// TIA Portal V20 export
ORGANIZATION_BLOCK "Startup"   // OB1000, LAD, Startup
TITLE = "Complete Restart"
AUTHOR : ERsystem_FA2_DH. Kim
// stored: AutoNumber false, IsIECCheckEnabled true, Namespace Unit1, SetENOAutomatically false
   VAR_INPUT
      LostRetentive : Bool;   // True if retentive data are lost
      LostRTC : Bool;   // True if date and time are lost
   END_VAR
   VAR_TEMP
      tempIndex : Int;   // Index of Unit in the array
   END_VAR
BEGIN

REGION Network 1: Unit Index Number
   // Assign the number of the unit to a temp for correct array index access.
   // Number is defined in PLC tags of Software Unit Global.
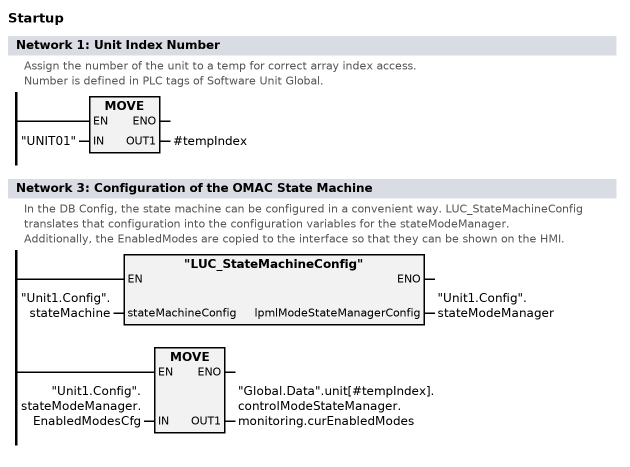
   RUNG wire#powerrail
      Move(in := "UNIT01", out1 => #tempIndex)
   END_RUNG
   // the same network as SCL:
   #tempIndex := "UNIT01";
END_REGION

REGION Network 2 (SCL): Build the Absolut Reference Designator
   // Set the Absoult Reference Designator in the DB Config. It is combined out of the parent reference designator and the own reference designator (=relative)
   IF LEN(IN := "Unit1.Config".unit.referenceDesignator.parent) <> 0 THEN
     "Unit1.Config".unit.referenceDesignator.combined := CONCAT_WSTRING(IN1 := "Unit1.Config".unit.referenceDesignator.parent, IN2 := WSTRING#'.', IN3 := "Unit1.Config".unit.referenceDesignator.relative);
   ELSE
     "Unit1.Config".unit.referenceDesignator.combined := "Unit1.Config".unit.referenceDesignator.relative;
   END_IF;
END_REGION

REGION Network 3: Configuration of the OMAC State Machine
   // In the DB Config, the state machine can be configured in a convenient way. LUC_StateMachineConfig translates that configuration into the configuration variables for the stateModeManager.
   // Additionally, the EnabledModes are copied to the interface so that they can be shown on the HMI.
   RUNG wire#powerrail
      "LUC_StateMachineConfig"(stateMachineConfig := "Unit1.Config".stateMachine, lpmlModeStateManagerConfig => "Unit1.Config".stateModeManager)
   END_RUNG
   RUNG wire#powerrail
      Move(in := "Unit1.Config".stateModeManager.EnabledModesCfg, out1 => "Global.Data".unit[#tempIndex].controlModeStateManager.monitoring.curEnabledModes)
   END_RUNG
   // the same network as SCL:
   "LUC_StateMachineConfig"(stateMachineConfig := "Unit1.Config".stateMachine,
                           lpmlModeStateManagerConfig => "Unit1.Config".stateModeManager);
   "Global.Data".unit[#tempIndex].controlModeStateManager.monitoring.curEnabledModes := "Unit1.Config".stateModeManager.EnabledModesCfg;
END_REGION

REGION Network 4 (SCL): Configuration of Stack Light
   // undefined
   "Unit1.Config".signalStack.undefined.static.red := FALSE;
   "Unit1.Config".signalStack.undefined.static.yellow := FALSE;
   "Unit1.Config".signalStack.undefined.static.blue := FALSE;
   "Unit1.Config".signalStack.undefined.static.green := FALSE;
   "Unit1.Config".signalStack.undefined.static.horn := FALSE;
   "Unit1.Config".signalStack.undefined.static.white := FALSE;
   "Unit1.Config".signalStack.undefined.static.user1 := FALSE;
   "Unit1.Config".signalStack.undefined.static.user2 := FALSE;

   "Unit1.Config".signalStack.undefined.flashing.red := TRUE;
   "Unit1.Config".signalStack.undefined.flashing.yellow := FALSE;
   "Unit1.Config".signalStack.undefined.flashing.blue := FALSE;
   "Unit1.Config".signalStack.undefined.flashing.green := FALSE;
   "Unit1.Config".signalStack.undefined.flashing.horn := FALSE;
   "Unit1.Config".signalStack.undefined.flashing.white := FALSE;
   "Unit1.Config".signalStack.undefined.flashing.user1 := FALSE;
   "Unit1.Config".signalStack.undefined.flashing.user2 := FALSE;

   // clearing
   "Unit1.Config".signalStack.clearing.static.red := FALSE;
   "Unit1.Config".signalStack.clearing.static.yellow := FALSE;
   "Unit1.Config".signalStack.clearing.static.blue := FALSE;
   "Unit1.Config".signalStack.clearing.static.green := FALSE;
   "Unit1.Config".signalStack.clearing.static.horn := FALSE;
   "Unit1.Config".signalStack.clearing.static.white := FALSE;
   "Unit1.Config".signalStack.clearing.static.user1 := FALSE;
   "Unit1.Config".signalStack.clearing.static.user2 := FALSE;

   "Unit1.Config".signalStack.clearing.flashing.red := TRUE;
   "Unit1.Config".signalStack.clearing.flashing.yellow := FALSE;
   "Unit1.Config".signalStack.clearing.flashing.blue := FALSE;
   "Unit1.Config".signalStack.clearing.flashing.green := FALSE;
   "Unit1.Config".signalStack.clearing.flashing.horn := FALSE;
   "Unit1.Config".signalStack.clearing.flashing.white := FALSE;
   "Unit1.Config".signalStack.clearing.flashing.user1 := FALSE;
   "Unit1.Config".signalStack.clearing.flashing.user2 := FALSE;

   // stopped
   "Unit1.Config".signalStack.stopped.static.red := TRUE;
   "Unit1.Config".signalStack.stopped.static.yellow := FALSE;
   "Unit1.Config".signalStack.stopped.static.blue := FALSE;
   "Unit1.Config".signalStack.stopped.static.green := FALSE;
   "Unit1.Config".signalStack.stopped.static.horn := FALSE;
   "Unit1.Config".signalStack.stopped.static.white := FALSE;
   "Unit1.Config".signalStack.stopped.static.user1 := FALSE;
   "Unit1.Config".signalStack.stopped.static.user2 := FALSE;

   "Unit1.Config".signalStack.stopped.flashing.red := FALSE;
   "Unit1.Config".signalStack.stopped.flashing.yellow := FALSE;
   "Unit1.Config".signalStack.stopped.flashing.blue := FALSE;
   "Unit1.Config".signalStack.stopped.flashing.green := FALSE;
   "Unit1.Config".signalStack.stopped.flashing.horn := FALSE;
   "Unit1.Config".signalStack.stopped.flashing.white := FALSE;
   "Unit1.Config".signalStack.stopped.flashing.user1 := FALSE;
   "Unit1.Config".signalStack.stopped.flashing.user2 := FALSE;

   // starting
   "Unit1.Config".signalStack.starting.static.red := FALSE;
   "Unit1.Config".signalStack.starting.static.yellow := FALSE;
   "Unit1.Config".signalStack.starting.static.blue := FALSE;
   "Unit1.Config".signalStack.starting.static.green := TRUE;
   "Unit1.Config".signalStack.starting.static.horn := FALSE;
   "Unit1.Config".signalStack.starting.static.white := FALSE;
   "Unit1.Config".signalStack.starting.static.user1 := FALSE;
   "Unit1.Config".signalStack.starting.static.user2 := FALSE;

   "Unit1.Config".signalStack.starting.flashing.red := FALSE;
   "Unit1.Config".signalStack.starting.flashing.yellow := FALSE;
   "Unit1.Config".signalStack.starting.flashing.blue := FALSE;
   "Unit1.Config".signalStack.starting.flashing.green := FALSE;
   "Unit1.Config".signalStack.starting.flashing.horn := FALSE;
   "Unit1.Config".signalStack.starting.flashing.white := FALSE;
   "Unit1.Config".signalStack.starting.flashing.user1 := FALSE;
   "Unit1.Config".signalStack.starting.flashing.user2 := FALSE;

   // idle
   "Unit1.Config".signalStack.idle.static.red := FALSE;
   "Unit1.Config".signalStack.idle.static.yellow := FALSE;
   "Unit1.Config".signalStack.idle.static.blue := FALSE;
   "Unit1.Config".signalStack.idle.static.green := FALSE;
   "Unit1.Config".signalStack.idle.static.horn := FALSE;
   "Unit1.Config".signalStack.idle.static.white := FALSE;
   "Unit1.Config".signalStack.idle.static.user1 := FALSE;
   "Unit1.Config".signalStack.idle.static.user2 := FALSE;

   "Unit1.Config".signalStack.idle.flashing.red := FALSE;
   "Unit1.Config".signalStack.idle.flashing.yellow := FALSE;
   "Unit1.Config".signalStack.idle.flashing.blue := FALSE;
   "Unit1.Config".signalStack.idle.flashing.green := TRUE;
   "Unit1.Config".signalStack.idle.flashing.horn := FALSE;
   "Unit1.Config".signalStack.idle.flashing.white := FALSE;
   "Unit1.Config".signalStack.idle.flashing.user1 := FALSE;
   "Unit1.Config".signalStack.idle.flashing.user2 := FALSE;

   // suspended
   "Unit1.Config".signalStack.suspended.static.red := FALSE;
   "Unit1.Config".signalStack.suspended.static.yellow := TRUE;
   "Unit1.Config".signalStack.suspended.static.blue := FALSE;
   "Unit1.Config".signalStack.suspended.static.green := FALSE;
   "Unit1.Config".signalStack.suspended.static.horn := FALSE;
   "Unit1.Config".signalStack.suspended.static.white := FALSE;
   "Unit1.Config".signalStack.suspended.static.user1 := FALSE;
   "Unit1.Config".signalStack.suspended.static.user2 := FALSE;

   "Unit1.Config".signalStack.suspended.flashing.red := FALSE;
   "Unit1.Config".signalStack.suspended.flashing.yellow := FALSE;
   "Unit1.Config".signalStack.suspended.flashing.blue := FALSE;
   "Unit1.Config".signalStack.suspended.flashing.green := FALSE;
   "Unit1.Config".signalStack.suspended.flashing.horn := FALSE;
   "Unit1.Config".signalStack.suspended.flashing.white := FALSE;
   "Unit1.Config".signalStack.suspended.flashing.user1 := FALSE;
   "Unit1.Config".signalStack.suspended.flashing.user2 := FALSE;

   // execute
   "Unit1.Config".signalStack.execute.static.red := FALSE;
   "Unit1.Config".signalStack.execute.static.yellow := FALSE;
   "Unit1.Config".signalStack.execute.static.blue := FALSE;
   "Unit1.Config".signalStack.execute.static.green := TRUE;
   "Unit1.Config".signalStack.execute.static.horn := FALSE;
   "Unit1.Config".signalStack.execute.static.white := FALSE;
   "Unit1.Config".signalStack.execute.static.user1 := FALSE;
   "Unit1.Config".signalStack.execute.static.user2 := FALSE;

   "Unit1.Config".signalStack.execute.flashing.red := FALSE;
   "Unit1.Config".signalStack.execute.flashing.yellow := FALSE;
   "Unit1.Config".signalStack.execute.flashing.blue := FALSE;
   "Unit1.Config".signalStack.execute.flashing.green := FALSE;
   "Unit1.Config".signalStack.execute.flashing.horn := FALSE;
   "Unit1.Config".signalStack.execute.flashing.white := FALSE;
   "Unit1.Config".signalStack.execute.flashing.user1 := FALSE;
   "Unit1.Config".signalStack.execute.flashing.user2 := FALSE;

   // stopping
   "Unit1.Config".signalStack.stopping.static.red := TRUE;
   "Unit1.Config".signalStack.stopping.static.yellow := FALSE;
   "Unit1.Config".signalStack.stopping.static.blue := FALSE;
   "Unit1.Config".signalStack.stopping.static.green := FALSE;
   "Unit1.Config".signalStack.stopping.static.horn := FALSE;
   "Unit1.Config".signalStack.stopping.static.white := FALSE;
   "Unit1.Config".signalStack.stopping.static.user1 := FALSE;
   "Unit1.Config".signalStack.stopping.static.user2 := FALSE;

   "Unit1.Config".signalStack.stopping.flashing.red := FALSE;
   "Unit1.Config".signalStack.stopping.flashing.yellow := FALSE;
   "Unit1.Config".signalStack.stopping.flashing.blue := FALSE;
   "Unit1.Config".signalStack.stopping.flashing.green := FALSE;
   "Unit1.Config".signalStack.stopping.flashing.horn := FALSE;
   "Unit1.Config".signalStack.stopping.flashing.white := FALSE;
   "Unit1.Config".signalStack.stopping.flashing.user1 := FALSE;
   "Unit1.Config".signalStack.stopping.flashing.user2 := FALSE;

   // aborting
   "Unit1.Config".signalStack.aborting.static.red := FALSE;
   "Unit1.Config".signalStack.aborting.static.yellow := FALSE;
   "Unit1.Config".signalStack.aborting.static.blue := FALSE;
   "Unit1.Config".signalStack.aborting.static.green := FALSE;
   "Unit1.Config".signalStack.aborting.static.horn := FALSE;
   "Unit1.Config".signalStack.aborting.static.white := FALSE;
   "Unit1.Config".signalStack.aborting.static.user1 := FALSE;
   "Unit1.Config".signalStack.aborting.static.user2 := FALSE;

   "Unit1.Config".signalStack.aborting.flashing.red := TRUE;
   "Unit1.Config".signalStack.aborting.flashing.yellow := FALSE;
   "Unit1.Config".signalStack.aborting.flashing.blue := FALSE;
   "Unit1.Config".signalStack.aborting.flashing.green := FALSE;
   "Unit1.Config".signalStack.aborting.flashing.horn := FALSE;
   "Unit1.Config".signalStack.aborting.flashing.white := FALSE;
   "Unit1.Config".signalStack.aborting.flashing.user1 := FALSE;
   "Unit1.Config".signalStack.aborting.flashing.user2 := FALSE;

   // aborted
   "Unit1.Config".signalStack.aborted.static.red := FALSE;
   "Unit1.Config".signalStack.aborted.static.yellow := FALSE;
   "Unit1.Config".signalStack.aborted.static.blue := FALSE;
   "Unit1.Config".signalStack.aborted.static.green := FALSE;
   "Unit1.Config".signalStack.aborted.static.horn := FALSE;
   "Unit1.Config".signalStack.aborted.static.white := FALSE;
   "Unit1.Config".signalStack.aborted.static.user1 := FALSE;
   "Unit1.Config".signalStack.aborted.static.user2 := FALSE;

   "Unit1.Config".signalStack.aborted.flashing.red := TRUE;
   "Unit1.Config".signalStack.aborted.flashing.yellow := FALSE;
   "Unit1.Config".signalStack.aborted.flashing.blue := FALSE;
   "Unit1.Config".signalStack.aborted.flashing.green := FALSE;
   "Unit1.Config".signalStack.aborted.flashing.horn := FALSE;
   "Unit1.Config".signalStack.aborted.flashing.white := FALSE;
   "Unit1.Config".signalStack.aborted.flashing.user1 := FALSE;
   "Unit1.Config".signalStack.aborted.flashing.user2 := FALSE;

   // holding
   "Unit1.Config".signalStack.holding.static.red := FALSE;
   "Unit1.Config".signalStack.holding.static.yellow := FALSE;
   "Unit1.Config".signalStack.holding.static.blue := FALSE;
   "Unit1.Config".signalStack.holding.static.green := FALSE;
   "Unit1.Config".signalStack.holding.static.horn := FALSE;
   "Unit1.Config".signalStack.holding.static.white := FALSE;
   "Unit1.Config".signalStack.holding.static.user1 := FALSE;
   "Unit1.Config".signalStack.holding.static.user2 := FALSE;

   "Unit1.Config".signalStack.holding.flashing.red := FALSE;
   "Unit1.Config".signalStack.holding.flashing.yellow := FALSE;
   "Unit1.Config".signalStack.holding.flashing.blue := TRUE;
   "Unit1.Config".signalStack.holding.flashing.green := FALSE;
   "Unit1.Config".signalStack.holding.flashing.horn := FALSE;
   "Unit1.Config".signalStack.holding.flashing.white := FALSE;
   "Unit1.Config".signalStack.holding.flashing.user1 := FALSE;
   "Unit1.Config".signalStack.holding.flashing.user2 := FALSE;

   // held
   "Unit1.Config".signalStack.held.static.red := FALSE;
   "Unit1.Config".signalStack.held.static.yellow := FALSE;
   "Unit1.Config".signalStack.held.static.blue := TRUE;
   "Unit1.Config".signalStack.held.static.green := FALSE;
   "Unit1.Config".signalStack.held.static.horn := FALSE;
   "Unit1.Config".signalStack.held.static.white := FALSE;
   "Unit1.Config".signalStack.held.static.user1 := FALSE;
   "Unit1.Config".signalStack.held.static.user2 := FALSE;

   "Unit1.Config".signalStack.held.flashing.red := FALSE;
   "Unit1.Config".signalStack.held.flashing.yellow := FALSE;
   "Unit1.Config".signalStack.held.flashing.blue := FALSE;
   "Unit1.Config".signalStack.held.flashing.green := FALSE;
   "Unit1.Config".signalStack.held.flashing.horn := FALSE;
   "Unit1.Config".signalStack.held.flashing.white := FALSE;
   "Unit1.Config".signalStack.held.flashing.user1 := FALSE;
   "Unit1.Config".signalStack.held.flashing.user2 := FALSE;

   // unholding
   "Unit1.Config".signalStack.unholding.static.red := FALSE;
   "Unit1.Config".signalStack.unholding.static.yellow := FALSE;
   "Unit1.Config".signalStack.unholding.static.blue := FALSE;
   "Unit1.Config".signalStack.unholding.static.green := TRUE;
   "Unit1.Config".signalStack.unholding.static.horn := FALSE;
   "Unit1.Config".signalStack.unholding.static.white := FALSE;
   "Unit1.Config".signalStack.unholding.static.user1 := FALSE;
   "Unit1.Config".signalStack.unholding.static.user2 := FALSE;

   "Unit1.Config".signalStack.unholding.flashing.red := FALSE;
   "Unit1.Config".signalStack.unholding.flashing.yellow := FALSE;
   "Unit1.Config".signalStack.unholding.flashing.blue := FALSE;
   "Unit1.Config".signalStack.unholding.flashing.green := FALSE;
   "Unit1.Config".signalStack.unholding.flashing.horn := FALSE;
   "Unit1.Config".signalStack.unholding.flashing.white := FALSE;
   "Unit1.Config".signalStack.unholding.flashing.user1 := FALSE;
   "Unit1.Config".signalStack.unholding.flashing.user2 := FALSE;

   // suspending
   "Unit1.Config".signalStack.suspending.static.red := FALSE;
   "Unit1.Config".signalStack.suspending.static.yellow := FALSE;
   "Unit1.Config".signalStack.suspending.static.blue := FALSE;
   "Unit1.Config".signalStack.suspending.static.green := FALSE;
   "Unit1.Config".signalStack.suspending.static.horn := FALSE;
   "Unit1.Config".signalStack.suspending.static.white := FALSE;
   "Unit1.Config".signalStack.suspending.static.user1 := FALSE;
   "Unit1.Config".signalStack.suspending.static.user2 := FALSE;

   "Unit1.Config".signalStack.suspending.flashing.red := FALSE;
   "Unit1.Config".signalStack.suspending.flashing.yellow := TRUE;
   "Unit1.Config".signalStack.suspending.flashing.blue := FALSE;
   "Unit1.Config".signalStack.suspending.flashing.green := FALSE;
   "Unit1.Config".signalStack.suspending.flashing.horn := FALSE;
   "Unit1.Config".signalStack.suspending.flashing.white := FALSE;
   "Unit1.Config".signalStack.suspending.flashing.user1 := FALSE;
   "Unit1.Config".signalStack.suspending.flashing.user2 := FALSE;

   // unsuspending
   "Unit1.Config".signalStack.unsuspending.static.red := FALSE;
   "Unit1.Config".signalStack.unsuspending.static.yellow := FALSE;
   "Unit1.Config".signalStack.unsuspending.static.blue := FALSE;
   "Unit1.Config".signalStack.unsuspending.static.green := TRUE;
   "Unit1.Config".signalStack.unsuspending.static.horn := FALSE;
   "Unit1.Config".signalStack.unsuspending.static.white := FALSE;
   "Unit1.Config".signalStack.unsuspending.static.user1 := FALSE;
   "Unit1.Config".signalStack.unsuspending.static.user2 := FALSE;

   "Unit1.Config".signalStack.unsuspending.flashing.red := FALSE;
   "Unit1.Config".signalStack.unsuspending.flashing.yellow := FALSE;
   "Unit1.Config".signalStack.unsuspending.flashing.blue := FALSE;
   "Unit1.Config".signalStack.unsuspending.flashing.green := FALSE;
   "Unit1.Config".signalStack.unsuspending.flashing.horn := FALSE;
   "Unit1.Config".signalStack.unsuspending.flashing.white := FALSE;
   "Unit1.Config".signalStack.unsuspending.flashing.user1 := FALSE;
   "Unit1.Config".signalStack.unsuspending.flashing.user2 := FALSE;

   // resetting
   "Unit1.Config".signalStack.resetting.static.red := TRUE;
   "Unit1.Config".signalStack.resetting.static.yellow := FALSE;
   "Unit1.Config".signalStack.resetting.static.blue := FALSE;
   "Unit1.Config".signalStack.resetting.static.green := FALSE;
   "Unit1.Config".signalStack.resetting.static.horn := FALSE;
   "Unit1.Config".signalStack.resetting.static.white := FALSE;
   "Unit1.Config".signalStack.resetting.static.user1 := FALSE;
   "Unit1.Config".signalStack.resetting.static.user2 := FALSE;

   "Unit1.Config".signalStack.resetting.flashing.red := FALSE;
   "Unit1.Config".signalStack.resetting.flashing.yellow := FALSE;
   "Unit1.Config".signalStack.resetting.flashing.blue := FALSE;
   "Unit1.Config".signalStack.resetting.flashing.green := FALSE;
   "Unit1.Config".signalStack.resetting.flashing.horn := FALSE;
   "Unit1.Config".signalStack.resetting.flashing.white := FALSE;
   "Unit1.Config".signalStack.resetting.flashing.user1 := FALSE;
   "Unit1.Config".signalStack.resetting.flashing.user2 := FALSE;

   // completing
   "Unit1.Config".signalStack.completing.static.red := FALSE;
   "Unit1.Config".signalStack.completing.static.yellow := FALSE;
   "Unit1.Config".signalStack.completing.static.blue := FALSE;
   "Unit1.Config".signalStack.completing.static.green := TRUE;
   "Unit1.Config".signalStack.completing.static.horn := FALSE;
   "Unit1.Config".signalStack.completing.static.white := FALSE;
   "Unit1.Config".signalStack.completing.static.user1 := FALSE;
   "Unit1.Config".signalStack.completing.static.user2 := FALSE;

   "Unit1.Config".signalStack.completing.flashing.red := FALSE;
   "Unit1.Config".signalStack.completing.flashing.yellow := FALSE;
   "Unit1.Config".signalStack.completing.flashing.blue := FALSE;
   "Unit1.Config".signalStack.completing.flashing.green := FALSE;
   "Unit1.Config".signalStack.completing.flashing.horn := FALSE;
   "Unit1.Config".signalStack.completing.flashing.white := FALSE;
   "Unit1.Config".signalStack.completing.flashing.user1 := FALSE;
   "Unit1.Config".signalStack.completing.flashing.user2 := FALSE;

   // completed
   "Unit1.Config".signalStack.completed.static.red := TRUE;
   "Unit1.Config".signalStack.completed.static.yellow := FALSE;
   "Unit1.Config".signalStack.completed.static.blue := FALSE;
   "Unit1.Config".signalStack.completed.static.green := FALSE;
   "Unit1.Config".signalStack.completed.static.horn := FALSE;
   "Unit1.Config".signalStack.completed.static.white := FALSE;
   "Unit1.Config".signalStack.completed.static.user1 := FALSE;
   "Unit1.Config".signalStack.completed.static.user2 := FALSE;

   "Unit1.Config".signalStack.completed.flashing.red := FALSE;
   "Unit1.Config".signalStack.completed.flashing.yellow := FALSE;
   "Unit1.Config".signalStack.completed.flashing.blue := FALSE;
   "Unit1.Config".signalStack.completed.flashing.green := FALSE;
   "Unit1.Config".signalStack.completed.flashing.horn := FALSE;
   "Unit1.Config".signalStack.completed.flashing.white := FALSE;
   "Unit1.Config".signalStack.completed.flashing.user1 := FALSE;
   "Unit1.Config".signalStack.completed.flashing.user2 := FALSE;
END_REGION
END_ORGANIZATION_BLOCK
